// TwinCAT 3 PLC project Example
// ProgramVersion: 3.1.4026.16
// libraries:
//   Tc2_Standard, * (Beckhoff Automation GmbH)
//   Tc2_System, * (Beckhoff Automation GmbH)
//   Tc2_Utilities, * (Beckhoff Automation GmbH)
//   VisuDialogs, * (System)
//   StageCore, * (_)
//   StageUtils, * (_)
// project tree:
//   / GlobalTextList.TcGTLO, PlcTask.TcTTO (not stored), Visualization Manager.TcVMO (not stored), VISU_TASK.TcTTO (not stored)
//   Heating/Ctx/ Heating_Ctx_Hmi.TcPOU, Heating_Ctx_Io.TcDUT (not stored), Heating_Ctx_Priv.TcPOU, Heating_Ctx_States.TcPOU
//   Heating/Ctx/Io/ Heating_Ctx_Io_In.TcDUT, Heating_Ctx_Io_Out.TcDUT (not stored)
//   Heating/ Heating.TcPOU, Heating_Ctx.TcPOU (not stored)
//   Heating/Receivers/ Heating_OnRequest.TcPOU
//   Heating/State/ Heating_State.TcPOU, Heating_State_Enabled.TcPOU, Heating_State_Disabled.TcPOU, Heating_State_Heatup.TcPOU, Heating_State_HeatingRoom.TcPOU, Heating_State_Safety.TcPOU, Heating_State_Fault.TcPOU
//   MAIN/ CST.TcGVL, COL.TcGVL, MAIN.TcPOU, MAIN.TcVIS, SIM.TcGVL
//   MAIN/SIM/ SimulationGlobalParameters.TcDUT, Tick.TcPOU, ValveSim.TcPOU
//   Room/Rooms/ ReceptionRoom.TcPOU, BaseRoom.TcPOU, StandardRoom.TcPOU
//   Room/ IArgToIRoom.TcPOU (not stored), I_Room.TcIO (not stored), Room_Ctx.TcPOU
//   Room/Ctx/ Room_Ctx_Hmi.TcPOU, Room_Ctx_Io.TcDUT, Room_Ctx_Priv.TcPOU (not stored), Room_Ctx_States.TcPOU
//   Room/Receivers/ Room_OnSystemEvent.TcPOU
//   Room/State/DemandHeating/ Room_State_DemandHeating.TcPOU, Room_State_DemandHeating_Hmi.TcPOU (not stored)
//   Room/State/LowTemperature/ Room_State_LowTemperature_Hmi.TcPOU (not stored), Room_State_LowTemperature.TcPOU
//   Room/State/ _Room_State.TcPOU, Room_State_Idle.TcPOU, Room_State_Fault.TcPOU, Room_State_Disabled.TcPOU
//   Room/UI/ Room_UiLogic.TcPOU
//   Safety/ Safety.TcPOU, Safety_Hmi.TcPOU
//   _UI/ UI_Heating.TcVIS, UI_Safety.TcVIS, UI_Room.TcVIS, UI_Sim.TcVIS, UI_Temp.TcVIS, UI_Demand.TcVIS (not stored)
// (motion and I/O tree: see PLC project stageutils)
// real-time tasks:
//   TASK Example: cycle T#10ms, priority 20, ADS port 350
//   TASK Test: cycle T#10ms, priority 21, ADS port 351
//   TASK VISU_TASK: cycle T#200000us, priority 30, ADS port 352

// ---- Heating/Ctx/Io/Heating_Ctx_Io_In.TcDUT
TYPE Heating_Ctx_Io_In :
STRUCT
	bPumpOverload	: BOOL;
	bBurnerOverload	: BOOL;
	
	rBoilerTemp		: REAL;
	rBoilerPressure	: REAL;
END_STRUCT
END_TYPE

// ---- MAIN/SIM/SimulationGlobalParameters.TcDUT
TYPE SimulationGlobalParameters :
STRUCT
	// Simulation parameter
	nTick							: UDINT := 1000; // ms
	bToggleSim						: BOOL;	

	// Heating system parameters
	rSystemTemperatureRisePerBurner	: REAL := 2.00;   // degC/tick
	rSystemTemperatureDropPassive	: LREAL := -0.01;  // degC/tick
	rSystemTemperatureDropPerHeater	: LREAL := -0.01;  // degC/tick per heater
	
	bToggleSystemTemperatureRise	: BOOL := FALSE;
	rSystemTemperatureRise			: LREAL := 0.2;
	
	bToggleSystemTemperatureFall	: BOOL := FALSE;
	rSystemTemperatureFall			: LREAL := 0.2;
	
	bToggleSystemPressureRise		: BOOL := FALSE;
	rSystemPressureRise				: LREAL := 0.10;   // bar/tick
	
	bToggleSystemPressureFall		: BOOL := FALSE;
	rSystemPressureFall				: LREAL := -0.10;   // bar/tick
	
	// Room parameters
	rRoomTemperaturePassiveDrop		: LREAL := -0.05;  // degC/tick
	rRoomTemperatureRisePerHeater	: LREAL := 0.50;   // degC/tick
	
	// Valve fault
	bToggleValveFault				: BOOL;
	
END_STRUCT
END_TYPE

// ---- Room/Ctx/Room_Ctx_Io.TcDUT
TYPE Room_Ctx_Io :
STRUCT
	bOpenValves			: BOOL;
END_STRUCT
END_TYPE

// ---- MAIN/CST.TcGVL
{attribute 'qualified_only'}
VAR_GLOBAL CONSTANT
	MAX_ROOM		: UDINT := 15;
	MAX_ESTOP		: UDINT := 2;
END_VAR

// ---- MAIN/COL.TcGVL
{attribute 'qualified_only'}
VAR_GLOBAL CONSTANT
{warning disable C0228}	// Disable warning: No initial value for variable ...
	RED			: Color(255, 0, 0, 255);
	BLACK		: Color(0, 0, 0, 255);
	ORANGE		: Color(255, 160, 0, 255);
	WHITE		: Color(255, 255, 255, 255);
	INVISIBLE	: Color(0, 0, 0, 0);
{warning restore C0228}
END_VAR

// ---- MAIN/SIM.TcGVL
{attribute 'qualified_only'}
VAR_GLOBAL PERSISTENT
	param			: SimulationGlobalParameters;
END_VAR

VAR_GLOBAL
	bTick				: BOOL;	

	rSystemTemperature	: REAL := 60;
	rSystemPressure		: REAL := 1;
	bFlow				: BOOL;
END_VAR

// ---- Heating/Ctx/Heating_Ctx_Hmi.TcPOU
FUNCTION_BLOCK Heating_Ctx_Hmi
VAR_INPUT
	sStatusText				: Str;
	sErrorText				: Str;
	nStatusColor			: Color;
	
	bButton					: BOOL;
	sButtonText				: Str;
	nButtonColor			: Color;	
END_VAR
VAR_OUTPUT PERSISTENT
	rMaxPressure			: REAL := 2.0; // bar
	rMinPressure			: REAL := 0.2; // bar
	
	rMaxTemperature			: REAL := 65.0; // °C
	rStdTemperature			: REAL := 60.0; // °C
	rMinTemperature			: REAL := 55.0; // °C
END_VAR

END_FUNCTION_BLOCK

// ---- Heating/Ctx/Heating_Ctx_Priv.TcPOU
FUNCTION_BLOCK Heating_Ctx_Priv
VAR_INPUT
	iActiveRoom		: I_Room;
END_VAR
VAR_OUTPUT
	iOnEnable		: I_SignalEmit;
	
	iQueue			: I_MutArgQueue;
END_VAR

END_FUNCTION_BLOCK

// ---- Heating/Ctx/Heating_Ctx_States.TcPOU
FUNCTION_BLOCK Heating_Ctx_States
VAR_OUTPUT
	iMgr			: I_StateManager;
	
	iSafety			: I_State;
	iFault			: I_State;
	iDisable		: I_State;
	iEnable			: I_State;
	iPump			: I_State;
	iHeatup			: I_State;
	
END_VAR

END_FUNCTION_BLOCK

// ---- Heating/Heating.TcPOU
FUNCTION_BLOCK Heating 
VAR_GENERIC CONSTANT
	ROOM_CAP		: UDINT := 20;
END_VAR

IMPLEMENTS I_Execute, I_Init
VAR_INPUT
	bPumpOverload	: BOOL;
	bBurnerOverload	: BOOL;

	rBoilerTemp		: LREAL := 60;
	rBoilerPressure	: LREAL := 1;
END_VAR
VAR_OUTPUT
	bPump			: BOOL;
	bBurner			: BOOL;
END_VAR
VAR
	_init			: Init(THIS^);
	_exe			: Execute(THIS^);
	_ctx			: Heating_Ctx;
	_tonPump		: TON;
	_tonBurner		: TON;	

	_entityStart	: EntityStart;
	_tag			: Tag := (Option := 'Heating');

	_smgr			: StateManager := (Proxy := _ctx.state.iMgr);
	
	_disabled		: Heating_State_Disabled(_ctx) := (Proxy := _ctx.state.iDisable);
	_safety         : Heating_State_Safety(_ctx) := (Proxy := _ctx.state.iSafety);
	_fault          : Heating_State_Fault(_ctx) := (Proxy := _ctx.state.iFault);
	_enabled        : Heating_State_Enabled(_ctx) := (Proxy := _ctx.state.iEnable);
	_pumping        : Heating_State_HeatingRoom(_ctx) := (Proxy := _ctx.state.iHeating);
	_heatup         : Heating_State_Heatup(_ctx) := (Proxy := _ctx.state.iHeatup);

	_enableEvent	: Signal := (Proxy := _ctx.priv.iOnEnable);
	_onRequestCall	: Heating_OnRequest(_ctx);
	_onRequest		: Receiver(_onRequestCall);
	
	_queue			: ArgQueue<ROOM_CAP> := (MutProxy := _ctx.priv.iQueue);
	
	_entityEnd		: EntityEnd;
END_VAR

METHOD Execute
VAR_INPUT
	nPhase: INT := 0;
END_VAR
// Inputs
_ctx.io.in.bBurnerOverload := bBurnerOverload;
_ctx.io.in.bPumpOverload := bPumpOverload;
_ctx.io.in.rBoilerPressure := rBoilerPressure;
_ctx.io.in.rBoilerTemp := rBoilerTemp;

// Outputs
_tonPump(IN := _ctx.io.out.bPump, PT := T#2S, Q => bPump);
_tonBurner(IN := _ctx.io.out.bBurner, PT := T#2S, Q => bBurner);

// SIMULATION

IF NOT sim.bTick THEN
	RETURN;
END_IF

// System temperature
IF bBurner THEN
	sim.rSystemTemperature := sim.rSystemTemperature + Sim.param.rSystemTemperatureRisePerBurner * Math.Random();
END_IF
sim.rSystemTemperature := sim.rSystemTemperature + Sim.param.rSystemTemperatureDropPassive * Math.Random();

IF sim.param.bToggleSystemTemperatureRise THEN
	sim.rSystemTemperature := sim.rSystemTemperature + Sim.param.rSystemTemperatureRise;
END_IF
IF sim.param.bToggleSystemTemperatureFall THEN
	sim.rSystemTemperature := sim.rSystemTemperature + Sim.param.rSystemTemperatureFall;
END_IF

IF sim.rSystemTemperature < 0 THEN
	sim.rSystemTemperature := 0;
ELSIF sim.rSystemTemperature > 100 THEN
	sim.rSystemTemperature := 100;
END_IF

sim.bFlow := bPump;

// System Pressure
IF sim.param.bToggleSystemPressureRise THEN
	sim.rSystemPressure := sim.rSystemPressure + Sim.param.rSystemPressureRise;
END_IF
IF sim.param.bToggleSystemPressureFall THEN
	sim.rSystemPressure := sim.rSystemPressure + Sim.param.rSystemPressureFall;
END_IF

IF sim.rSystemPressure < 0 THEN
	sim.rSystemPressure := 0;
ELSIF sim.rSystemPressure > 10 THEN
	sim.rSystemPressure := 10;
END_IF

// Write IO

rBoilerTemp := sim.rSystemTemperature;
rBoilerPressure := sim.rSystemPressure;
END_METHOD

METHOD Init
VAR_INPUT
	nPhase: INT;
END_VAR
_smgr.Request(_disabled);
END_METHOD

END_FUNCTION_BLOCK

// ---- Heating/State/Heating_State_Disabled.TcPOU
FUNCTION_BLOCK Heating_State_Disabled EXTENDS Heating_State
VAR_INPUT
END_VAR
VAR_OUTPUT
END_VAR
VAR
END_VAR

METHOD PROTECTED OnEntry
_ctx.hmi.sStatusText := 'Heating disabled!';
_ctx.hmi.nStatusColor := COL.BLACK.Raw;

_ctx.hmi.sButtonText := 'Press to ENABLE!';
_ctx.hmi.nButtonColor := COL.BLACK.Raw;

_ctx.io.out.bBurner := FALSE;
_ctx.io.out.bPump := FALSE;

_ctx.priv.iQueue.Clear();
END_METHOD

METHOD PROTECTED OnExecute
IF _ctx.hmi.bButton THEN
	_ctx.hmi.bButton := FALSE;
	_ctx.state.iMgr.Request(_ctx.state.iEnable);
END_IF
END_METHOD

END_FUNCTION_BLOCK

// ---- Heating/State/Heating_State.TcPOU
FUNCTION_BLOCK ABSTRACT Heating_State EXTENDS State
VAR
	_ctx			: REFERENCE TO Heating_Ctx;
END_VAR

(*FB_Init is always available implicitly and it is used primarily for initialization.
The return value is not evaluated. For a specific influence, you can also declare the
methods explicitly and provide additional code there with the standard initialization
code. You can evaluate the return value.*)
METHOD FB_Init : BOOL
VAR_INPUT
	(* TRUE: the retain variables are initialized (reset warm / reset cold)*)
	bInitRetains	: BOOL;
	(* TRUE: the instance will be copied to the copy code afterward (online change)*)
	bInCopyCode	: BOOL;
	iEntity	: Core.I_Entity;
	ctx		: REFERENCE TO Heating_Ctx;
END_VAR
_ctx REF= ctx;
END_METHOD

END_FUNCTION_BLOCK

// ---- Heating/State/Heating_State_Safety.TcPOU
FUNCTION_BLOCK Heating_State_Safety EXTENDS Heating_State IMPLEMENTS I_Callable, I_Init
VAR
	_init					: Init(THIS^);
	_safetyRec				: Receiver(THIS^);
	_bSafetyStopActive			: BOOL;
END_VAR

METHOD Call
VAR_INPUT
	iArg		: StageCore.I_Arg;
END_VAR
VAR
	_iSafeModeOn: I_BoolArg;
END_VAR
IF IsOk(IArgToIBoolArg(iArg, _iSafeModeOn)) THEN
	IF _iSafeModeOn.Get THEN
		_bSafetyStopActive := TRUE;
		_ctx.state.iMgr.Request(_ctx.state.iSafety);
	ELSE
		_bSafetyStopActive := FALSE;
		_ctx.state.iMgr.Request(_ctx.state.iDisable);
	END_IF
END_IF
END_METHOD

METHOD PROTECTED CanDeactivate : BOOL
CanDeactivate := NOT _bSafetyStopActive;
END_METHOD

METHOD Init
VAR_INPUT
	nPhase: INT;
END_VAR
VAR
	i			: Iter(1);
	_r			: Result;
	
	_iEntity	: I_Entity;
	_iSignal	: I_Signal;
	
	
END_VAR
WHILE IsOk(GetEntity(i.Next(), _iEntity)) DO
	IF IsOk(GetSignal(_iEntity, '*._safetyEvent', _iSignal)) THEN
		IF IsFail(_iSignal.Pair(_safetyRec), nOut => _r) THEN
			DebugMsg(_iSignal, CONCAT('Could not be paired! Error code: ', TO_STRING(_r)));
		END_IF
		
		RETURN;
	END_IF
END_WHILE

DebugMsg(THIS^, CONCAT('_safetyRec not paired! Error code: ', TO_STRING(_r)));
END_METHOD

METHOD PROTECTED OnEntry
_ctx.hmi.sStatusText := 'Safety engaged! Check safety system...';
_ctx.hmi.nStatusColor := COL.RED.Raw;

_ctx.hmi.sButtonText := '';
_ctx.hmi.nButtonColor := COL.INVISIBLE.Raw;

_ctx.io.out.bBurner := FALSE;
_ctx.io.out.bPump := FALSE;

_ctx.priv.iQueue.Clear();
END_METHOD

END_FUNCTION_BLOCK

// ---- Safety/Safety.TcPOU
FUNCTION_BLOCK Safety 
VAR_GENERIC CONSTANT
	ESTOP_CAP		: UDINT := 2;
END_VAR
IMPLEMENTS I_Execute
VAR_INPUT
	bSafetyOk		: BOOL;
	bEStopActive	: ARRAY[1..ESTOP_CAP] OF BOOL;
END_VAR
VAR_OUTPUT
	bSafetyRun		: BOOL;
	bErrAck			: BOOL;
END_VAR
VAR
	_exe			: Execute(THIS^);
	_hmi			: Safety_Hmi<ESTOP_CAP>;
	_nStep			: USINT;
	_tonTimeout		: TON;	

	_entityStart		: EntityStart;
	_tag				: Tag := (Option := 'Safety');

	_safetyEvent		: Signal;
	_bSafetyStopActive	: BoolArg(FALSE);
	
	_entityEnd			: EntityEnd;
END_VAR

METHOD Execute
VAR_INPUT
	nPhase: INT;
END_VAR
VAR
	i			: UDINT;
END_VAR
FOR i := 1 TO ESTOP_CAP DO
	_hmi.bEStopActive[i] := bESTopActive[i];
END_FOR


CASE _nStep OF
	0: // Fault Init
		_bSafetyStopActive.OpSet(TRUE);
		_safetyEvent.Emit(_bSafetyStopActive);
		bSafetyRun	:= FALSE;
		
		_nStep := 1;
		
		_hmi.bHideReset := TRUE;
		_hmi.nStatusColor := COL.RED.Raw;
		_hmi.sStatusText := 'Safety Stop Activated!';

	1: // Fault
		_hmi.bHideReset := NOT bSafetyOk;
		IF bSafetyOk AND _hmi.bReset THEN
			_hmi.bReset := FALSE;
			
			_nStep := 2;
		END_IF

	2: // Reset init
		bSafetyRun	:= TRUE;
		
		_nStep		:= 3;
		
		_hmi.bHideReset := TRUE;
		_hmi.nStatusColor := COL.RED.Raw;
		_hmi.sStatusText := 'Reset in progress...';
		
	3: // Reset
	
		bErrAck		:= TRUE;
		
		_tonTimeout(IN := TRUE, PT := T#5S);
		
		IF bSafetyOk THEN
			_tonTimeout(IN := FALSE);
			_nStep := 4;
		ELSIF _tonTimeout.Q THEN
			_tonTimeout(IN := FALSE);
			_nStep := 0;
		END_IF	

	4:	// Op Init
		bErrAck		:= FALSE;
	
		_bSafetyStopActive.OpSet(FALSE);
		_safetyEvent.Emit(_bSafetyStopActive);
		_nStep := 5;
		
		_hmi.bHideReset := TRUE;
		_hmi.nStatusColor := COL.BLACK.Raw;
		_hmi.sStatusText := 'Safety OK!';

	5:	// Op
		IF NOT bSafetyOk THEN
			_nStep := 0;
		END_IF
END_CASE
END_METHOD

END_FUNCTION_BLOCK

// ---- Safety/Safety_Hmi.TcPOU
FUNCTION_BLOCK Safety_Hmi
VAR_GENERIC CONSTANT
	ESTOP_CAP		: UDINT := 4;
END_VAR

VAR_INPUT
	bEStopActive	: ARRAY[1..ESTOP_CAP] OF BOOL;
	
	sStatusText		: Str;
	nStatusColor	: Color;
	
	bReset			: BOOL;
	bHideReset		: BOOL;
END_VAR

END_FUNCTION_BLOCK

// ---- Heating/State/Heating_State_Fault.TcPOU
FUNCTION_BLOCK Heating_State_Fault EXTENDS Heating_State IMPLEMENTS I_Execute
VAR
	_exe		: Execute(THIS^);
END_VAR

METHOD Execute
VAR_INPUT
	nPhase: INT;
END_VAR
VAR
	cmp			: TagCmp;
	bFault		: BOOL;
END_VAR
IF _ctx.io.in.bBurnerOverload THEN
	bFault := TRUE;
END_IF

IF _ctx.io.in.bPumpOverload THEN
	bFault := TRUE;
END_IF

IF _ctx.io.in.rBoilerPressure > _ctx.hmi.rMaxPressure THEN
	bFault := TRUE;
END_IF

IF _ctx.io.in.rBoilerPressure < _ctx.hmi.rMinPressure THEN
	bFault := TRUE;
END_IF

IF _ctx.io.in.rBoilerTemp > _ctx.hmi.rMaxTemperature THEN
	bFault := TRUE;
END_IF

IF cmp.Set(_ctx.state.iMgr.Current.Tag).Match(_ctx.state.iFault.Tag).Match(_ctx.state.iSafety.Tag).IsTrue() THEN
	bFault := FALSE;
END_IF

IF NOT bFault THEN
	RETURN;
END_IF

_ctx.state.iMgr.Request(_ctx.state.iFault);
END_METHOD

METHOD PROTECTED OnEntry
IF _ctx.io.in.bBurnerOverload THEN
	_ctx.hmi.sErrorText := 'Caused by burner overload!';
ELSIF _ctx.io.in.bPumpOverload THEN
	_ctx.hmi.sErrorText := 'Caused by pump overload!';
ELSIF _ctx.io.in.rBoilerPressure > _ctx.hmi.rMaxPressure THEN
	_ctx.hmi.sErrorText := 'Caused by boiler overpressure!';
ELSIF _ctx.io.in.rBoilerPressure < _ctx.hmi.rMinPressure THEN
	_ctx.hmi.sErrorText := 'Caused by boiler underpressure!';
ELSIF _ctx.io.in.rBoilerTemp > _ctx.hmi.rMaxTemperature THEN
	_ctx.hmi.sErrorText := 'Caused by boiler overheat!';
END_IF

_ctx.hmi.sStatusText := CONCAT('Fault: ', _ctx.hmi.sErrorText);

_ctx.hmi.nStatusColor := COL.RED.Raw;

_ctx.hmi.sButtonText := 'Press to RESET';
_ctx.hmi.nButtonColor := COL.INVISIBLE.Raw;

_ctx.io.out.bBurner := FALSE;
_ctx.io.out.bPump := FALSE;

_ctx.priv.iQueue.Clear();
END_METHOD

METHOD PROTECTED OnExecute
VAR
	bFault : BOOL;
END_VAR
IF _ctx.io.in.bBurnerOverload THEN
	bFault := TRUE;
END_IF

IF _ctx.io.in.bPumpOverload THEN
	bFault := TRUE;;
END_IF

IF _ctx.io.in.rBoilerPressure > _ctx.hmi.rMaxPressure THEN
	bFault := TRUE;;
END_IF

IF _ctx.io.in.rBoilerPressure < _ctx.hmi.rMinPressure THEN
	bFault := TRUE;;
END_IF

IF _ctx.io.in.rBoilerTemp > _ctx.hmi.rMaxTemperature THEN
	bFault := TRUE;;
END_IF

IF _ctx.hmi.bButton AND NOT bFault THEN
	_ctx.hmi.bButton := FALSE;
	_ctx.state.iMgr.Request(_ctx.state.iDisable);
ELSIF NOT bFault THEN
	_ctx.hmi.nButtonColor := COL.BLACK.Raw;	
ELSE
	_ctx.hmi.nButtonColor := COL.INVISIBLE.Raw;	
	_ctx.hmi.bButton := FALSE;
END_IF
END_METHOD

END_FUNCTION_BLOCK

// ---- Heating/State/Heating_State_Enabled.TcPOU
FUNCTION_BLOCK Heating_State_Enabled EXTENDS Heating_State
VAR_INPUT
END_VAR
VAR_OUTPUT
END_VAR
VAR
END_VAR

METHOD PROTECTED OnEntry
_ctx.hmi.sStatusText := 'Heating enabled: Waiting for requests...';
_ctx.hmi.nStatusColor := COL.BLACK.Raw;

_ctx.hmi.sButtonText := 'Press to DISABLE!';
_ctx.hmi.nButtonColor := COL.BLACK.Raw;

_ctx.io.out.bBurner := FALSE;
_ctx.io.out.bPump := FALSE;

IF _ctx.state.iMgr.Current = _ctx.state.iDisable THEN
	_ctx.priv.iOnEnable.Emit();
END_IF
END_METHOD

METHOD PROTECTED OnExecute
VAR
	_iRoomArg		: I_Arg;
END_VAR
IF _ctx.hmi.bButton THEN
	_ctx.hmi.bButton := FALSE;
	_ctx.state.iMgr.Request(_ctx.state.iDisable);
	
ELSIF _ctx.io.in.rBoilerTemp < _ctx.hmi.rMinTemperature THEN
	_ctx.state.iMgr.Request(_ctx.state.iHeatup);
	
ELSIF IsOk(_ctx.priv.iQueue.Pop(iArg => _iRoomArg)) THEN
	IF IsOk(IArgToIRoom(_iRoomArg, iDest => _ctx.priv.iActiveRoom)) THEN
		IF _ctx.priv.iActiveRoom.IsActive THEN
			_ctx.state.iMgr.Request(_ctx.state.iHeating);
		END_IF
	ELSE
		_ctx.hmi.sErrorText := 'Room Queue - Incorrect iRoomArg!';
	END_IF
END_IF
END_METHOD

END_FUNCTION_BLOCK

// ---- Heating/State/Heating_State_HeatingRoom.TcPOU
FUNCTION_BLOCK Heating_State_HeatingRoom EXTENDS Heating_State
VAR CONSTANT
	EXIT_STEP		: USINT := 7;
	READY_STEP		: USINT := 8;
END_VAR
VAR
	_nStep		: USINT;
	_tonTimeout	: TON;
	_sErrMsg	: Str;
	_iNextState : I_State;
END_VAR

METHOD PROTECTED CanActivate : BOOL
CanActivate :=  _ctx.state.iMgr.Current = _ctx.state.iEnable;
END_METHOD

METHOD PROTECTED OnEntry
VAR
	strb			: Strb;
END_VAR
_ctx.hmi.sStatusText := strb.Append('Heating enabled: Pumping to room ')
							.Append(UDINT_TO_STRING(_ctx.priv.iActiveRoom.Id))
							.Append('...')
							.Read();
							
_ctx.hmi.nStatusColor := COL.BLACK.Raw;

_ctx.hmi.sButtonText := 'Press to DISABLE!';
_ctx.hmi.nButtonColor := COL.BLACK.Raw;

_ctx.io.out.bBurner := FALSE;
_ctx.io.out.bPump := FALSE;

_nStep := 0;
_tonTimeout(IN := FALSE);

_iNextState := _ctx.state.iEnable;
END_METHOD

METHOD PROTECTED OnExecute
VAR
	strb		: Strb;
END_VAR
IF _ctx.priv.iActiveRoom = 0 THEN
	_iNextState := _ctx.state.iFault;	

	_nStep := EXIT_STEP;
	_ctx.hmi.sErrorText := 'HeatingRoom - Incorrect iActiveRoom value!';
ELSIF _ctx.hmi.bButton THEN
	_ctx.hmi.bButton := FALSE;
	_iNextState := _ctx.state.iDisable;
	
	_nStep := 4;
ELSIF _tonTimeout.Q THEN
	_ctx.priv.iActiveRoom.GoFault(strb.Set('Timeout on: ').Append(_sErrMsg).Read());
	
	_nStep := EXIT_STEP;
ELSIF _nStep < 4 AND_THEN NOT _ctx.priv.iActiveRoom.IsActive THEN
	_iNextState := _ctx.state.iEnable;	

	_nStep := 4;
END_IF

IF _ctx.priv.iActiveRoom <> 0 THEN
	_tonTimeout(IN := TRUE, PT := _ctx.priv.iActiveRoom.Timeout);
END_IF

CASE _nStep OF
	0:
		_sErrMsg := 'Valve opening!';
		_ctx.priv.iActiveRoom.GoHeat();
		_nStep := 1;
		
	1:
		IF _ctx.priv.iActiveRoom.IsOpen THEN
			_nStep := 2;
		END_IF
	2:	
		
		_ctx.io.out.bPump := TRUE;
		_nStep := 3;
	3:
		_sErrMsg := 'Heating!';
		IF _ctx.priv.iActiveRoom.IsReady THEN
			_nStep := 4;
		END_IF
	4:	
		_ctx.io.out.bPump := FALSE;
		_nStep := 5;
	5:
		_sErrMsg := 'Valve closing!';
		_ctx.priv.iActiveRoom.GoIdle();
		_nStep := 6;
	6:
		IF _ctx.priv.iActiveRoom.IsClosed THEN
			_nStep := EXIT_STEP;
		END_IF
	7:
		IF _iNextState <> 0 THEN
			_ctx.state.iMgr.Request(_iNextState);
		ELSE
			_ctx.hmi.sErrorText := 'HeatingRoom - Incorrect _iNextState value!';
			_ctx.state.iMgr.Request(_ctx.state.iFault);
		END_IF
		
		_nStep := READY_STEP;
END_CASE
END_METHOD

(*
Executed when the state transitions to another state.  
Provides a hook for defining cleanup or transition-specific behavior.
*)
METHOD PROTECTED OnExit
IF _ctx.priv.iActiveRoom <> 0 THEN
	_ctx.priv.iActiveRoom.GoIdle();
END_IF
END_METHOD

END_FUNCTION_BLOCK

// ---- Heating/State/Heating_State_Heatup.TcPOU
FUNCTION_BLOCK Heating_State_Heatup EXTENDS Heating_State
VAR_INPUT
END_VAR
VAR_OUTPUT
END_VAR
VAR
END_VAR

METHOD CanActivate : BOOL
CanActivate :=  _ctx.state.iMgr.Current = _ctx.state.iEnable;
END_METHOD

METHOD OnEntry
_ctx.hmi.sStatusText := 'Heating enabled: Heating up...';
_ctx.hmi.nStatusColor := COL.BLACK.Raw;

_ctx.hmi.sButtonText := 'Press to DISABLE!';
_ctx.hmi.nButtonColor := COL.BLACK.Raw;

_ctx.io.out.bBurner := TRUE;
_ctx.io.out.bPump := TRUE;
END_METHOD

METHOD OnExecute
IF _ctx.hmi.bButton THEN
	_ctx.hmi.bButton := FALSE;
	_ctx.state.iMgr.Request(_ctx.state.iDisable);
	
ELSIF _ctx.io.in.rBoilerTemp >= _ctx.hmi.rStdTemperature THEN
	_ctx.state.iMgr.Request(_ctx.state.iEnable);
END_IF
END_METHOD

END_FUNCTION_BLOCK

// ---- Heating/Receivers/Heating_OnRequest.TcPOU
FUNCTION_BLOCK Heating_OnRequest IMPLEMENTS I_Callable
VAR
	_ctx			: REFERENCE TO Heating_Ctx;
END_VAR

METHOD Call
VAR_INPUT
	iArg				: Core.I_Arg;
END_VAR
VAR
	_iRoom				: I_Room;
END_VAR
IF IsOk(IArgToIRoom(iArg, iDest => _iRoom)) THEN
	_ctx.priv.iQueue.Push(_iRoom);
END_IF
END_METHOD

//FB_Init is always available implicitly and it is used primarily for initialization.
//The return value is not evaluated. For a specific influence, you can also declare the
//methods explicitly and provide additional code there with the standard initialization
//code. You can evaluate the return value.
METHOD FB_Init: BOOL
VAR_INPUT
    bInitRetains: BOOL; // TRUE: the retain variables are initialized (reset warm / reset cold)
    bInCopyCode: BOOL;  // TRUE: the instance will be copied to the copy code afterward (online change)

	ctx			: REFERENCE TO Heating_Ctx;   
END_VAR
_ctx REF= ctx;
END_METHOD

END_FUNCTION_BLOCK

// ---- MAIN/MAIN.TcPOU
PROGRAM MAIN
VAR
	safety				: Safety<CST.MAX_ESTOP>;
	heating				: Heating<CST.MAX_ROOM>;
	
	stdRoom				: ARRAY[1..3] OF StandardRoom;
	reception			: ReceptionRoom;

	dbgInfo				: DebugInfo;
	rtTick				: R_TRIG;
END_VAR

rtTick(CLK :=  Tick(sim.param.nTick), Q => sim.bTick);
sim.bTick := sim.bTick AND sim.param.bToggleSim;

Runtime();

END_PROGRAM

// ---- Room/Rooms/StandardRoom.TcPOU
FUNCTION_BLOCK StandardRoom EXTENDS BaseRoom
VAR_INPUT
	rTemperature	: LREAL := 20.0 + Math.Random();
END_VAR
VAR    	
    // Entity
    _entityExtend	: EntityExtend(_entityStart);
	
    _lowTemperature : Room_State_LowTemperature(_ctx, rTemperature);
    _demand         : Room_State_DemandHeating(_ctx);
   
    _entityEnd2		: EntityEnd;
END_VAR

METHOD Execute
SUPER^.Execute();

// Simulation
IF NOT sim.bTick THEN
	RETURN;
END_IF

IF bInletValve AND bOutletValve THEN
	rTemperature := rTemperature + sim.param.rRoomTemperatureRisePerHeater * Math.Random();
END_IF

rTemperature := rTemperature + sim.param.rRoomTemperaturePassiveDrop * Math.Random();

IF rTemperature < 0 THEN
	rTemperature := 0;
ELSIF rTemperature > 100 THEN
	rTemperature := 100;
END_IF
END_METHOD

END_FUNCTION_BLOCK

// ---- Room/Rooms/BaseRoom.TcPOU
FUNCTION_BLOCK BaseRoom IMPLEMENTS I_Execute, I_Init
VAR_INPUT	
	bInletValveIsClosed	: BOOL;
	bInletValveIsOpen	: BOOL;
	
	bOutletValveIsClosed: BOOL;
	bOutletValveIsOpen	: BOOL;
END_VAR
VAR_OUTPUT
	bInletValve		: BOOL;
	bOutletValve	: BOOL;
END_VAR
VAR    
    // Initialization and execution logic
    _init           : Init(THIS^);
    _exe            : Execute(THIS^);
    _ctx            : Room_Ctx;
	
	// UI Logic
    _uiLogic        : Room_UiLogic(_ctx);
	
    // Simulation
    _inletSim       : ValveSim(bInletValve, bInletValveIsOpen, bInletValveIsClosed);
    _outletSim      : ValveSim(bOutletValve, bOutletValveIsOpen, bOutletValveIsClosed);	
	
	
    // Entity
    _entityStart    : EntityStart;
	
    _tag            : Tag := (Option := CONCAT('Room_', UDINT_TO_STRING(_ctx.Id)));
    
    // State Manager
    _smgr           : StateManager := (Proxy := _ctx.state.iMgr);
    
    // States
    _disabled       : Room_State_Disabled(_ctx) := (Proxy := _ctx.state.iDisable);
    _fault          : Room_State_Fault(_ctx) := (Proxy := _ctx.state.iFault);
    _idle           : Room_State_Idle(_ctx) := (Proxy := _ctx.state.iIdle);
	
	// Receiver
    _onSystemEvent  : Room_OnSystemEvent(_ctx);
    
    // Signal
    _requestEvent   : Signal := (Proxy := _ctx.priv.iRequestEvent);
   
    _entityEnd      : EntityEnd;
END_VAR

METHOD Execute
VAR_INPUT
	nPhase: INT;
END_VAR
// HMI

_ctx.hmi.sData := '';

// Inputs
_ctx.io.bValvesOpen := bInletValveIsOpen AND bOutletValveIsOpen;
_ctx.io.bValvesClosed := bInletValveIsClosed AND bOutletValveIsClosed;

// Outputs
bInletValve := _ctx.io.bOpenValves;
bOutletValve := _ctx.io.bOpenValves;

// Simulation
IF NOT sim.bTick THEN
	RETURN;
END_IF

IF bInletValve AND bOutletValve THEN
	sim.rSystemTemperature := sim.rSystemTemperature + sim.param.rSystemTemperatureDropPerHeater * Math.Random();
END_IF
END_METHOD

METHOD Init
VAR_INPUT
	nPhase: INT;
END_VAR
_smgr.Request(_idle);
END_METHOD

END_FUNCTION_BLOCK

// ---- Room/Room_Ctx.TcPOU
FUNCTION_BLOCK Room_Ctx
VAR_INPUT
	io		: Room_Ctx_Io; // different
	hmi		: Room_Ctx_Hmi; // the same
	state	: Room_Ctx_States; // the same
	priv	: Room_Ctx_Priv; // the same but different logic
END_VAR

END_FUNCTION_BLOCK

// ---- Room/Ctx/Room_Ctx_Hmi.TcPOU
FUNCTION_BLOCK Room_Ctx_Hmi
VAR_INPUT
	nId						: UDINT;	

	sStatusText				: Str;
	sErrorText				: Str;
	nStatusColor			: Color;
	
	sData					: Str;
	
	bDisable				: BOOL;
	sDisableText			: Str;
	
	bReset					: BOOL;
	bHideReset				: BOOL;
END_VAR
VAR_OUTPUT PERSISTENT
	nTimeout				: UDINT := 1;
END_VAR

END_FUNCTION_BLOCK

// ---- Room/Ctx/Room_Ctx_States.TcPOU
FUNCTION_BLOCK Room_Ctx_States
VAR_OUTPUT
	iMgr			: I_StateManager;
	
	iSystemOff		: I_State;
	iFault			: I_State;
	iDisable		: I_State;
	iIdle			: I_State;
END_VAR

END_FUNCTION_BLOCK

// ---- Room/UI/Room_UiLogic.TcPOU
FUNCTION_BLOCK Room_UiLogic IMPLEMENTS I_Execute
VAR_INPUT
END_VAR
VAR_OUTPUT
END_VAR
VAR
	_exe			: Execute(THIS^);
	_ctx			: REFERENCE TO Room_Ctx;
	
	_bPrvDisable	: BOOL;
END_VAR

METHOD Execute
IF _bPrvDisable <> _ctx.hmi.bDisable THEN
	_bPrvDisable := _ctx.hmi.bDisable;
	
	IF _ctx.hmi.bDisable THEN
		_ctx.hmi.sDisableText := 'Press to ENABLE!';
	ELSE
		_ctx.hmi.sDisableText := 'Press to DISABLE!';
	END_IF	
END_IF
END_METHOD

//FB_Init is always available implicitly and it is used primarily for initialization.
//The return value is not evaluated. For a specific influence, you can also declare the
//methods explicitly and provide additional code there with the standard initialization
//code. You can evaluate the return value.
METHOD FB_Init: BOOL
VAR_INPUT
    bInitRetains: BOOL; // TRUE: the retain variables are initialized (reset warm / reset cold)
    bInCopyCode: BOOL;  // TRUE: the instance will be copied to the copy code afterward (online change)
	
	ctx			: REFERENCE TO Room_Ctx;
END_VAR
_ctx REF= ctx;

IF _ctx.hmi.bDisable THEN
	_ctx.hmi.sDisableText := 'Press to ENABLE!';
ELSE
	_ctx.hmi.sDisableText := 'Press to DISABLE!';
END_IF
END_METHOD

END_FUNCTION_BLOCK

// ---- MAIN/SIM/ValveSim.TcPOU
FUNCTION_BLOCK ValveSim IMPLEMENTS I_Execute
VAR
	_bInput		: REFERENCE TO BOOL;	
	_bIsOpen	: REFERENCE TO BOOL;
	_bIsClosed	: REFERENCE TO BOOL;	

	_exe		: Execute(THIS^);
	_ton		: TON := (PT := LREAL_TO_TIME(Math.Random() * 1000));
	_rt			: R_TRIG;
	_ft			: F_TRIG;
	_bInit		: BOOL := TRUE;
END_VAR

(*
If registered, this method will be executed cyclically.
*)
METHOD Execute
VAR_INPUT
	nPhase: INT;
END_VAR
_rt(CLK := _bInput);
_ft(CLK := _bInput);
IF _rt.Q OR _ft.Q OR _bInit THEN
	_ton.IN := TRUE;
	_bInit := FALSE;
END_IF

_ton();
IF _ton.Q AND SIM.param.bToggleValveFault THEN
	_ton(IN := FALSE);
	_bIsClosed := FALSE;
	_bIsOpen := FALSE;
	SIM.param.bToggleValveFault := FALSE;
ELSIF _ton.Q AND _bInput THEN
	_ton(IN := FALSE);
	_bIsOpen := TRUE;
	_bIsClosed := FALSE;
ELSIF _ton.Q AND NOT _bInput THEN
	_ton(IN := FALSE);
	_bIsOpen := FALSE;
	_bIsClosed := TRUE;	
END_IF
END_METHOD

//FB_Init is always available implicitly and it is used primarily for initialization.
//The return value is not evaluated. For a specific influence, you can also declare the
//methods explicitly and provide additional code there with the standard initialization
//code. You can evaluate the return value.
METHOD FB_Init: BOOL
VAR_INPUT
    bInitRetains: BOOL; // TRUE: the retain variables are initialized (reset warm / reset cold)
    bInCopyCode: BOOL;  // TRUE: the instance will be copied to the copy code afterward (online change) 

  	bInput		: REFERENCE TO BOOL;	
	bIsOpen		: REFERENCE TO BOOL;
	bIsClosed	: REFERENCE TO BOOL;	
END_VAR
_bInput REF= bInput;
_bIsOpen REF= bIsOpen;
_bIsClosed REF= bIsClosed;
END_METHOD

END_FUNCTION_BLOCK

// ---- Room/State/Room_State_Disabled.TcPOU
FUNCTION_BLOCK Room_State_Disabled EXTENDS _Room_State
VAR_INPUT
END_VAR
VAR_OUTPUT
END_VAR
VAR
END_VAR

METHOD OnEntry
_ctx.io.bOpenValves := FALSE;

_ctx.priv.bActive := FALSE;
_ctx.priv.bReady := FALSE;

_ctx.hmi.sStatusText := 'ROOM DISABLED!';
_ctx.hmi.nStatusColor := COL.RED.Raw;

_ctx.hmi.bHideReset := TRUE;
END_METHOD

METHOD OnExecute
IF NOT _ctx.hmi.bDisable THEN
	_ctx.state.iMgr.Request(_ctx.state.iIdle);
END_IF
END_METHOD

END_FUNCTION_BLOCK

// ---- Room/State/_Room_State.TcPOU
FUNCTION_BLOCK ABSTRACT _Room_State EXTENDS State
VAR
	_ctx	: REFERENCE TO Room_Ctx;
END_VAR

(*FB_Init is always available implicitly and it is used primarily for initialization.
The return value is not evaluated. For a specific influence, you can also declare the
methods explicitly and provide additional code there with the standard initialization
code. You can evaluate the return value.*)
METHOD FB_Init : BOOL
VAR_INPUT
	(* TRUE: the retain variables are initialized (reset warm / reset cold)*)
	bInitRetains	: BOOL;
	(* TRUE: the instance will be copied to the copy code afterward (online change)*)
	bInCopyCode	: BOOL;
	iEntity	: Core.I_Entity;
	ctx		: REFERENCE TO Room_Ctx;
END_VAR
_ctx REF= ctx;
END_METHOD

END_FUNCTION_BLOCK

// ---- Room/State/Room_State_Fault.TcPOU
FUNCTION_BLOCK Room_State_Fault EXTENDS _Room_State
VAR_INPUT
END_VAR
VAR_OUTPUT
END_VAR
VAR
END_VAR

METHOD PROTECTED OnEntry
_ctx.io.bOpenValves := FALSE;

_ctx.priv.bActive := FALSE;
_ctx.priv.bReady := FALSE;

_ctx.hmi.sStatusText := CONCAT('Fault: ', _ctx.hmi.sErrorText);
_ctx.hmi.nStatusColor := COL.RED.Raw;

_ctx.hmi.bHideReset := FALSE;
END_METHOD

METHOD PROTECTED OnExecute
IF _ctx.hmi.bReset THEN
	_ctx.hmi.bReset := FALSE;
	
	_ctx.state.iMgr.Request(_ctx.state.iIdle);
END_IF
END_METHOD

METHOD PROTECTED OnExit
_ctx.hmi.sErrorText := 'Undefined';
END_METHOD

END_FUNCTION_BLOCK

// ---- Room/State/Room_State_Idle.TcPOU
FUNCTION_BLOCK Room_State_Idle EXTENDS _Room_State
VAR_INPUT
END_VAR
VAR_OUTPUT
END_VAR
VAR
END_VAR

METHOD OnEntry
_ctx.io.bOpenValves := FALSE;

_ctx.priv.bActive := FALSE;
_ctx.priv.bReady := FALSE;

_ctx.hmi.sStatusText := 'Heating ON: Idle';
_ctx.hmi.nStatusColor := COL.BLACK.Raw;

_ctx.hmi.bHideReset := TRUE;
END_METHOD

METHOD OnExecute
IF _ctx.hmi.bDisable THEN
	_ctx.state.iMgr.Request(_ctx.state.iDisable);
END_IF
END_METHOD

END_FUNCTION_BLOCK

// ---- Room/Receivers/Room_OnSystemEvent.TcPOU
FUNCTION_BLOCK Room_OnSystemEvent IMPLEMENTS I_Init, I_Callable
VAR
	_init				: Init(THIS^);
	_onSystemEvent		: Receiver(THIS^);
	
	_bError				: BOOL;
	
	_iResumeEvent		: I_Signal;
	_iPauseEvent		: I_Signal;
	_iEnableEvent		: I_Signal;
	_iDisableEvent		: I_Signal;
	
	_ctx				: REFERENCE TO Room_Ctx;
END_VAR

METHOD PRIVATE _GetSignalAndPair
VAR_INPUT
	iEntity		: I_Entity;
	sToFind		: Str;
END_VAR
VAR_OUTPUT
	iSignal	: I_Signal;
END_VAR
VAR
	_r			: Result;
	strb		: Strb;
END_VAR
CASE GetSignal(iEntity, sToFind, iSignal) OF
	Ok:
		IF IsFail(iSignal.Pair(_onSystemEvent), nOut => _r) THEN
			_bError := TRUE;
			DebugMsg(iSignal, strb.Append('Cannot pair _systemRec with this signal! Error code: ').Append(INT_TO_STRING(_r)).Read());
		END_IF
	ELSE
		_bError := TRUE;
		DebugMsg(THIS^, strb.Append('Cannot pair _systemRec with a ').Append(sToFind).Append('!').Read());
		DebugMsg(iEntity, strb.Append(sToFind).Append(' not found!').Read());
END_CASE
END_METHOD

METHOD Call
VAR_INPUT
	iArg	: StageCore.I_Arg;
END_VAR
VAR
	cmp		: TagCmp;
	_iTag	: I_Tag;
END_VAR
IF _bError THEN
	_ctx.hmi.sErrorText := 'Incorrect receiver initialization!';
	_ctx.state.iMgr.Request(_ctx.state.iFault);
	RETURN;
END_IF

IF IsErr(IArgToITag(iArg, _iTag)) THEN
	_ctx.hmi.sErrorText := 'Incorrect call argument!';
	_ctx.state.iMgr.Request(_ctx.state.iFault);
	RETURN;
END_IF

cmp.Set(_iTag);
IF cmp.Match(_iEnableEvent.Tag).IsTrue() THEN
	IF _ctx.state.iMgr.Current = 0 THEN
		RETURN;
	END_IF

	cmp.Set(_ctx.state.iMgr.Current.Tag);
	IF cmp.Match(_ctx.state.iFault.Tag)
			.Match(_ctx.state.iDisable.Tag)
			.Match(_ctx.state.iIdle.Tag)
			.IsTrue() THEN
			
		RETURN;
	END_IF
	
	_ctx.priv.iRequestEvent.Emit(_ctx);
	
	RETURN;
END_IF
END_METHOD

//FB_Init is always available implicitly and it is used primarily for initialization.
//The return value is not evaluated. For a specific influence, you can also declare the
//methods explicitly and provide additional code there with the standard initialization
//code. You can evaluate the return value.
METHOD FB_Init: BOOL
VAR_INPUT
    bInitRetains: BOOL; // TRUE: the retain variables are initialized (reset warm / reset cold)
    bInCopyCode: BOOL;  // TRUE: the instance will be copied to the copy code afterward (online change)
	
	ctx			: REFERENCE TO Room_Ctx;
END_VAR
_ctx REF= ctx;
END_METHOD

METHOD Init
VAR_INPUT
	nPhase: INT;
END_VAR
VAR
	i			: Iter(1);
	_iEntity	: I_Entity;
END_VAR
WHILE IsOk(GetEntity(i.Next(), _iEntity)) DO
	IF IsFail(HasTagOption(_iEntity, 'Heating')) THEN
		CONTINUE;
	END_IF
	
	_GetSignalAndPair(_iEntity, '*._enableEvent', iSignal => _iEnableEvent);
	
	RETURN;
END_WHILE
END_METHOD

END_FUNCTION_BLOCK

// ---- Room/State/LowTemperature/Room_State_LowTemperature.TcPOU
FUNCTION_BLOCK Room_State_LowTemperature EXTENDS _Room_State IMPLEMENTS I_Execute, I_Init
VAR
	_init					: Init(THIS^);
	_exe					: Execute(THIS^);
	_hmi					: Room_State_LowTemperature_Hmi;
	_rTemperature			: REFERENCE TO LREAL;
END_VAR

METHOD PROTECTED CanActivate : BOOL
CanActivate := _ctx.state.iMgr.Current = _ctx.state.iIdle;
END_METHOD

METHOD Execute
VAR_INPUT
	nPhase: INT;
END_VAR
VAR
	_iSelf		: I_State := THIS^;
	_strb		: strb;
END_VAR
_strb.Set(_ctx.hmi.sData)
		.Append(' ')
		.Append(Strf.Fmt('%0.2f', F_LReal(_rTemperature)))
		.Append(' degC');

_ctx.hmi.sData := _strb.Read();

IF _ctx.state.iMgr.Current <> _ctx.state.iIdle THEN
	RETURN;
END_IF

IF _ctx.state.iMgr.Current = _iSelf THEN
	RETURN;
END_IF

IF _rTemperature < _hmi.rLowTemperature THEN
	_ctx.state.iMgr.Request(THIS^);
END_IF
END_METHOD

(*FB_Init is always available implicitly and it is used primarily for initialization.
The return value is not evaluated. For a specific influence, you can also declare the
methods explicitly and provide additional code there with the standard initialization
code. You can evaluate the return value.*)
METHOD FB_Init : BOOL
VAR_INPUT
	(* TRUE: the retain variables are initialized (reset warm / reset cold)*)
	bInitRetains	: BOOL;
	(* TRUE: the instance will be copied to the copy code afterward (online change)*)
	bInCopyCode	: BOOL;
	ctx				: REFERENCE TO Room_Ctx;
	rTemperature	: REFERENCE TO LREAL;
END_VAR
_rTemperature REF= rTemperature;
END_METHOD

METHOD Init
VAR_INPUT
	nPhase: INT;
END_VAR
VAR
	i			: Iter(1);
	_iEntity	: I_Entity;
	_iRec		: I_Receiver;
	_r			: Result;
	strb		: Strb;
END_VAR
WHILE IsOk(GetEntity(i.Next(), _iEntity)) DO
	IF IsNone(HasTagOption(_iEntity, 'Heating')) THEN
		CONTINUE;
	END_IF
	
	IF IsOk(GetReceiver(_iEntity, '*._onRequest', _iRec)) THEN
		IF IsErr(_ctx.priv.iRequestEvent.Pair(_iRec), nOut => _r) THEN
			DebugMsg(_iRec, strb.Append('Cannot pair _onRequest with this receiver! Error code: ').Append(TO_STRING(_r)).Read());
		END_IF
		
		RETURN;
	END_IF
END_WHILE

DebugMsg(THIS^, strb.Append('Cannot pair _requestEvent with a ').Append('_onRequest').Append('!').Read());
DebugMsg(_iEntity, strb.Append('_onRequest').Append(' not found!').Read());
END_METHOD

METHOD PROTECTED OnEntry
_ctx.io.bOpenValves := FALSE;

_ctx.priv.bActive := TRUE;
_ctx.priv.bReady := FALSE;

_ctx.hmi.sStatusText := 'Heating ON: Low Temperature...';
_ctx.hmi.nStatusColor := COL.BLACK.Raw;

_ctx.hmi.bHideReset := TRUE;

_ctx.priv.iRequestEvent.Emit(_ctx);
END_METHOD

METHOD PROTECTED OnExecute
IF _ctx.hmi.bDisable THEN
	_ctx.state.iMgr.Request(_ctx.state.iDisable);
ELSIF _rTemperature >= _hmi.rHighTemperature THEN
	_ctx.priv.bReady := TRUE;
END_IF
END_METHOD

END_FUNCTION_BLOCK

// ---- Room/State/DemandHeating/Room_State_DemandHeating.TcPOU
FUNCTION_BLOCK Room_State_DemandHeating EXTENDS _Room_State IMPLEMENTS I_Execute
VAR
	_exe				: Execute(THIS^);
	_hmi				: Room_State_DemandHeating_Hmi;
	_tonActive			: TON;
END_VAR

METHOD PROTECTED CanActivate : BOOL
CanActivate := _ctx.state.iMgr.Current = _ctx.state.iIdle;
END_METHOD

METHOD Execute
VAR_INPUT
	nPhase: INT;
END_VAR
VAR
	_iSelf		: I_State := THIS^;
	_strb		: Strb;
END_VAR
_strb.Set(_ctx.hmi.sData)
		.Append(' On: ').Append(strf.SimpleTime(_tonActive.ET, 'S', 'M'));

_ctx.hmi.sData := _strb.Read();

IF _ctx.state.iMgr.Current <> _ctx.state.iIdle THEN
	RETURN;
END_IF

IF _ctx.state.iMgr.Current = _iSelf THEN
	RETURN;
END_IF

IF _hmi.bDemandButton THEN
	_ctx.state.iMgr.Request(THIS^);
END_IF
END_METHOD

METHOD Init
VAR
	i			: Iter(1);
	_iEntity	: I_Entity;
	_iRec		: I_Receiver;
	_r			: Result;
	strb		: Strb;
END_VAR
WHILE IsOk(GetEntity(i.Next(), _iEntity)) DO
	IF IsNone(HasTagOption(_iEntity, 'Heating')) THEN
		CONTINUE;
	END_IF
	
	IF IsOk(GetReceiver(_iEntity, '*._onRequest', _iRec)) THEN
		IF IsErr(_ctx.priv.iRequestEvent.Pair(_iRec), nOut => _r) THEN
			DebugMsg(_iRec, strb.Append('Cannot pair _onRequest with this receiver! Error code: ').Append(TO_STRING(_r)).Read());
		END_IF
		
		RETURN;
	END_IF
END_WHILE

DebugMsg(THIS^, strb.Append('Cannot pair _requestEvent with a ').Append('_onRequest').Append('!').Read());
DebugMsg(_iEntity, strb.Append('_onRequest').Append(' not found!').Read());
END_METHOD

METHOD PROTECTED OnEntry
_ctx.io.bOpenValves := FALSE;

_ctx.priv.bActive := TRUE;
_ctx.priv.bReady := FALSE;

_ctx.hmi.sStatusText := 'Heating ON: Scheduled demand...';
_ctx.hmi.nStatusColor := COL.BLACK.Raw;

_ctx.hmi.bHideReset := TRUE;

_tonActive(IN := FALSE);

_ctx.priv.iRequestEvent.Emit(_ctx);
END_METHOD

METHOD PROTECTED OnExecute
_tonActive(IN := _ctx.io.bValvesOpen, PT := UDINT_TO_TIME(_hmi.nActivationTime * 1000));
IF _ctx.hmi.bDisable THEN
	_ctx.state.iMgr.Request(_ctx.state.iDisable);
ELSIF NOT _hmi.bDemandButton THEN
	_ctx.priv.bReady := TRUE;
ELSIF _tonActive.Q THEN
	_ctx.priv.bReady := TRUE;
	_hmi.bDemandButton := FALSE;
END_IF
END_METHOD

METHOD PROTECTED OnExit
VAR_INPUT
END_VAR
_hmi.bDemandButton := FALSE;
END_METHOD

END_FUNCTION_BLOCK

// ---- Room/Rooms/ReceptionRoom.TcPOU
FUNCTION_BLOCK ReceptionRoom EXTENDS BaseRoom
VAR_INPUT
	rTemperature	: LREAL := 20.0 + Math.Random();
END_VAR
VAR    
    // Entity
    _entityExtend	: EntityExtend(_entityStart);
	
    _lowTemperature	: Room_State_LowTemperature(_ctx, rTemperature);
	
    _entityEnd2		: EntityEnd;
END_VAR

METHOD Execute
VAR_INPUT
	nPhase: INT;
END_VAR
SUPER^.Execute(nPhase);

// Simulation
IF NOT sim.bTick THEN
	RETURN;
END_IF

IF bInletValve AND bOutletValve THEN
	rTemperature := rTemperature + sim.param.rRoomTemperatureRisePerHeater * Math.Random();
END_IF

rTemperature := rTemperature + sim.param.rRoomTemperaturePassiveDrop * Math.Random();

IF rTemperature < 0 THEN
	rTemperature := 0;
ELSIF rTemperature > 100 THEN
	rTemperature := 100;
END_IF
END_METHOD

END_FUNCTION_BLOCK

// ---- MAIN/SIM/Tick.TcPOU
FUNCTION Tick : BOOL
VAR_INPUT
	nTimeInMs	: ULINT;
	nTaskInMs	: ULINT := 20;
END_VAR

Tick := (GetSysTime() MOD (nTimeInMs * 10_000)) < (nTaskInMs * 10_000);

END_FUNCTION

// ---- GlobalTextList.TcGTLO
TEXTLIST GlobalTextList
  443 = '%.2f'
  858 = '%2.2f'
  701 = '%2.2f bar'
  165 = '%2.2f bar/tick'
  1000 = '%2.2f min'
  388 = '%2.2f s'
  181 = '%2.2f °C'
  899 = '%2.2f °C/tick'
  252 = '%i'
  752 = '%i min'
  296 = '%i s'
  862 = '%s'
  231 = 'Active'
  553 = 'Auto Sim'
  595 = 'Burner'
  999 = 'Burner Overload'
  870 = 'Click to change'
  18 = 'Demand'
  819 = 'Demand Activation Time'
  935 = 'Demand Active'
  969 = 'Drain Outlet Open'
  754 = 'Drain Outlet Valve Open'
  445 = 'Drain Speed: %.4f'
  336 = 'Enable Switch'
  958 = 'Enable Tank Switch'
  520 = 'EStop Button'
  707 = 'Feedback Ok'
  476 = 'Fill Speed: %.4f'
  923 = 'Filling Timeout:'
  698 = 'Filling Timeout: %s'
  393 = 'Heating'
  226 = 'Heating:'
  371 = 'High Level: %.2f'
  140 = 'High Level: %s'
  42 = 'High Temperature'
  254 = 'hmi.sMultiButtonText'
  89 = 'Level Sensor'
  616 = 'Low Level: %.2f'
  234 = 'Low Level: %s'
  738 = 'Low Temperature'
  762 = 'Max Pressure'
  409 = 'Max Pressure:'
  676 = 'Max Temp.'
  397 = 'Max Temp.:'
  731 = 'Mid Temp.'
  67 = 'Mid Temp.:'
  141 = 'Min Pressure'
  32 = 'Min Pressure:'
  630 = 'Min Temp.'
  441 = 'Min Temp.:'
  700 = 'NoWater'
  848 = 'OFF Delay'
  934 = 'ON delay'
  998 = 'Overload'
  728 = 'PASSIVE HEATING'
  116 = 'Press to Reset'
  342 = 'Pump'
  317 = 'Pump Overload'
  190 = 'Request Button'
  261 = 'Request Level: %.2f'
  452 = 'Request Level: %s'
  160 = 'Reset Output'
  106 = 'Room'
  64 = 'RoomTemperaturePassiveDrop'
  649 = 'RoomTemperatureRisePerHeater'
  111 = 'rRoomTemperaturePassiveDrop'
  468 = 'rRoomTemperatureRisePerHeater'
  142 = 'rSystemPressureFall'
  531 = 'rSystemPressureRise'
  247 = 'rSystemTemperatureDropPassive'
  485 = 'rSystemTemperatureDropPerHeater'
  498 = 'rSystemTemperatureFall'
  155 = 'rSystemTemperatureRise'
  173 = 'rSystemTemperatureRisePerBurner'
  305 = 'Run Output'
  300 = 'RunPump'
  489 = 'Safety'
  684 = 'Safety Ok'
  444 = 'Safety Run'
  517 = 'SafetyOk'
  629 = 'Simulation'
  411 = 'State:'
  587 = 'State: %s'
  664 = 'Status:'
  233 = 'Status: %s'
  471 = 'Sys. Pressure.'
  974 = 'Sys. Pressure.:'
  548 = 'Sys. Temp.'
  446 = 'Sys. Temp.:'
  338 = 'System Operational'
  534 = 'SystemPressureFall'
  450 = 'SystemPressureRise'
  420 = 'SystemTemperatureDropPassive'
  410 = 'SystemTemperatureDropPerHeater'
  648 = 'SystemTemperatureFall'
  264 = 'SystemTemperatureRise'
  918 = 'SystemTemperatureRisePerBurner'
  12 = 'Tank 0'
  237 = 'Tank 1'
  741 = 'Tank 2'
  288 = 'Tank 3'
  262 = 'Tick'
  743 = 'Timeout'
  737 = 'Timeout: %.2f'
  430 = 'Timeout: %s'
  596 = 'Toggle'
  315 = 'ToggleValveFault'
  379 = 'ToggleValveFault - Next valve action will fail'
  1064 = 'ToggleValveFault - Next valve actuation will fail'
  168 = 'TriggerValveFault'
END_TEXTLIST

// ---- MAIN/MAIN.TcVIS
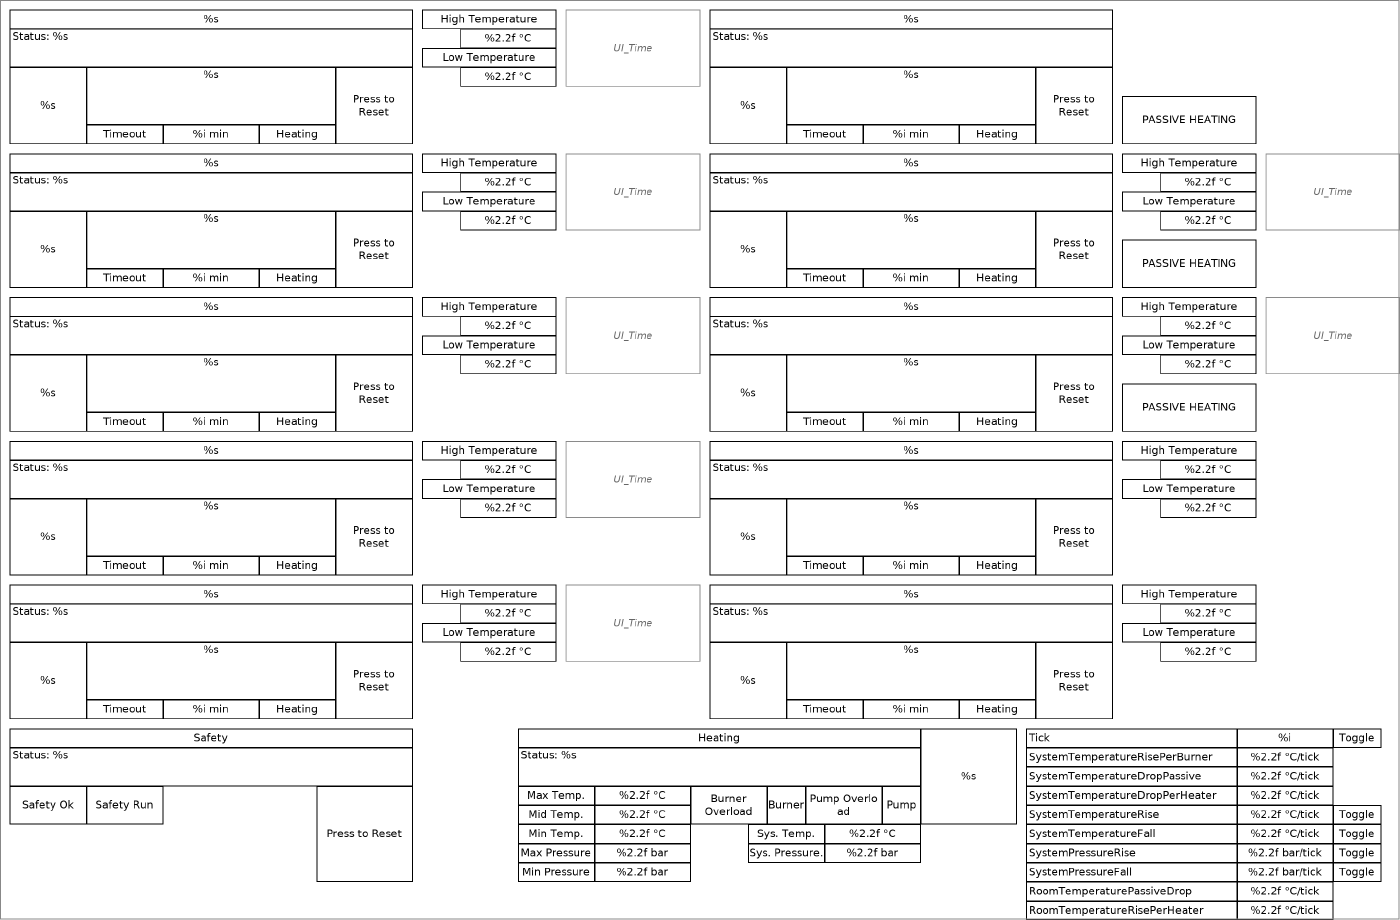
VISUALIZATION MAIN  // 1460x960
    Frame (10,760 520x100)
        shows UI_Safety(pou := MAIN.safety)
    Frame (540,760 520x160)
        shows UI_Heating(pou := MAIN.heating)
    Frame (10,10 420x140)
        shows UI_Room(ctx := MAIN.standardRoom[1]._ctx)
    Frame (10,160 420x140)
        shows UI_Room(ctx := MAIN.standardRoom[2]._ctx)
    Frame (10,310 420x140)
        shows UI_Room(ctx := MAIN.standardRoom[3]._ctx)
    Frame (10,460 420x140)
        shows UI_Room(ctx := MAIN.standardRoom[4]._ctx)
    Frame (10,610 420x140)
        shows UI_Room(ctx := MAIN.standardRoom[5]._ctx)
    Frame (440,10 140x80)
        shows UI_Temp(setting := MAIN.standardRoom[1]._settings.temp)
    Frame (440,160 140x80)
        shows UI_Temp(setting := MAIN.standardRoom[2]._settings.temp)
    Frame (440,310 140x80)
        shows UI_Temp(setting := MAIN.standardRoom[3]._settings.temp)
    Frame (440,460 140x80)
        shows UI_Temp(setting := MAIN.standardRoom[4]._settings.temp)
    Frame (440,610 140x80)
        shows UI_Temp(setting := MAIN.standardRoom[5]._settings.temp)
    Frame (740,10 420x140)
        shows UI_Room(ctx := MAIN.receptionRoom._ctx)
    Frame (740,160 420x140)
        shows UI_Room(ctx := MAIN.conferentionRoom01._ctx)
    Frame (740,310 420x140)
        shows UI_Room(ctx := MAIN.conferentionRoom02._ctx)
    Frame (740,460 420x140)
        shows UI_Room(ctx := MAIN.storeRoom01._ctx)
    Frame (740,610 420x140)
        shows UI_Room(ctx := MAIN.storeRoom02._ctx)
    Frame (1170,160 140x80)
        shows UI_Temp(setting := MAIN.conferentionRoom01._settings.temp)
    Frame (1170,310 140x80)
        shows UI_Temp(setting := MAIN.conferentionRoom02._settings.temp)
    Frame (1170,460 140x80)
        shows UI_Temp(setting := MAIN.storeRoom01._settings)
    Frame (1170,610 140x80)
        shows UI_Temp(setting := MAIN.storeRoom02._settings)
    Frame (1320,160 140x80)
        shows UI_Time(settings := MAIN.conferentionRoom01._settings.timee)
    Frame (590,10 140x80)
        shows UI_Time(settings := MAIN.standardRoom[1]._settings.timee)
    Frame (590,160 140x80)
        shows UI_Time(settings := MAIN.standardRoom[2]._settings.timee)
    Frame (590,310 140x80)
        shows UI_Time(settings := MAIN.standardRoom[3]._settings.timee)
    Frame (590,610 140x80)
        shows UI_Time(settings := MAIN.standardRoom[5]._settings.timee)
    Frame (590,460 140x80)
        shows UI_Time(settings := MAIN.standardRoom[4]._settings.timee)
    Frame (1320,310 140x80)
        shows UI_Time(settings := MAIN.conferentionRoom02._settings.timee)
    Rectangle (1170,400 140x50), "PASSIVE HEATING", colour toggle: MAIN.conferentionRoom02._settings.bEnablePassive
        toggle MAIN.conferentionRoom02._settings.bEnablePassive
    Rectangle (1170,250 140x50), "PASSIVE HEATING", colour toggle: MAIN.conferentionRoom01._settings.bEnablePassive
        toggle MAIN.conferentionRoom01._settings.bEnablePassive
    Rectangle (1170,100 140x50), "PASSIVE HEATING"
        toggle MAIN.receptionRoom._bEnablePassive
    Frame (1070,760 370x200)
        shows UI_Sim(param := SIM.param)
END_VISUALIZATION

// ---- _UI/UI_Heating.TcVIS
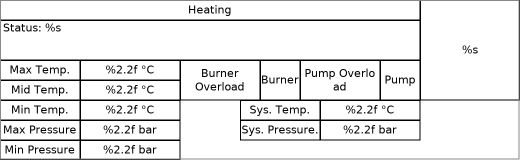
VISUALIZATION UI_Heating  // 520x160
VAR_IN_OUT
	pou			: Heating<CST.MAX_ROOM>;
END_VAR
VAR
END_VAR
    Rectangle (0,0 420x20), "Heating"
    Rectangle (0,20 420x40), "Status: %s", text variable: pou._ctx.hmi.sStatusText
        p55702900: pou._ctx.hmi.nStatusColor
    Rectangle (420,0 100x100), "%s", text variable: pou._ctx.hmi.sButtonText
        p55702900: pou._ctx.hmi.nButtonColor
        toggle pou._ctx.hmi.bButton
    Rectangle (0,60 80x20), "Max Temp."
    Rectangle (0,80 80x20), "Mid Temp."
    Rectangle (0,100 80x20), "Min Temp."
    Rectangle (80,60 100x20), "%2.2f °C", text variable: pou._ctx.hmi.rMaxTemperature
        OnMouseClick: write the text variable via Default
    Rectangle (80,80 100x20), "%2.2f °C", text variable: pou._ctx.hmi.rStdTemperature
        OnMouseClick: write the text variable via Default
    Rectangle (80,100 100x20), "%2.2f °C", text variable: pou._ctx.hmi.rMinTemperature
        OnMouseClick: write the text variable via Default
    Rectangle (0,140 80x20), "Min Pressure"
    Rectangle (0,120 80x20), "Max Pressure"
    Rectangle (80,120 100x20), "%2.2f bar", text variable: pou._ctx.hmi.rMaxPressure
        OnMouseClick: write the text variable via Default
    Rectangle (80,140 100x20), "%2.2f bar", text variable: pou._ctx.hmi.rMinPressure
        OnMouseClick: write the text variable via Default
    Rectangle (380,60 40x40), "Pump", colour toggle: pou.bPump
        toggle pou.bPump
    Rectangle (260,60 40x40), "Burner", colour toggle: pou.bBurner
        toggle pou.bBurner
    Rectangle (300,60 80x40), "Pump Overload", colour toggle: pou.bPumpOverload
        toggle pou.bPumpOverload
    Rectangle (180,60 80x40), "Burner Overload", colour toggle: pou.bBurnerOverload
        toggle pou.bBurnerOverload
    Rectangle (320,120 100x20), "%2.2f bar", text variable: pou.rBoilerPressure
    Rectangle (240,100 80x20), "Sys. Temp."
    Rectangle (240,120 80x20), "Sys. Pressure."
    Rectangle (320,100 100x20), "%2.2f °C", text variable: pou.rBoilerTemp
END_VISUALIZATION

// ---- _UI/UI_Safety.TcVIS
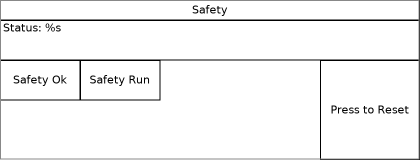
VISUALIZATION UI_Safety  // 420x160
VAR_IN_OUT
	pou			: Safety<CST.MAX_ESTOP>;
END_VAR
    Rectangle (0,0 420x20), "Safety"
    Rectangle (0,20 420x40), "Status: %s", text variable: pou._hmi.sStatusText
        p55702900: pou._hmi.nStatusColor
    Rectangle (320,60 100x100), "Press to Reset", invisible if: pou._hmi.bHideReset
        toggle pou._hmi.bReset
    Rectangle (0,60 80x40), "Safety Ok", colour toggle: pou.bSafetyOk
        toggle pou.bSafetyOk
    Rectangle (80,60 80x40), "Safety Run", colour toggle: pou.bSafetyRun
        toggle pou.bSafetyRun
END_VISUALIZATION

// ---- _UI/UI_Room.TcVIS
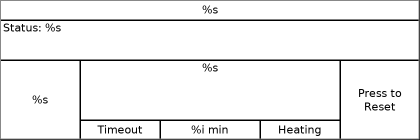
VISUALIZATION UI_Room  // 420x140
VAR_IN_OUT
	ctx			: Room_Ctx;
END_VAR
    Rectangle (0,0 420x20), "%s", text variable: CONCAT('Room ', UDINT_TO_STRING(ctx.hmi.nId))
    Rectangle (0,20 420x40), "Status: %s", text variable: ctx.hmi.sStatusText
        p55702900: ctx.hmi.nStatusColor
    Rectangle (0,60 80x80), "%s", text variable: ctx.hmi.sDisableText
        toggle ctx.hmi.bDisable
    Rectangle (340,60 80x80), "Press to Reset", invisible if: ctx.hmi.bHideReset
        toggle ctx.hmi.bReset
    Rectangle (80,60 260x60), "%s", text variable: ctx.hmi.sData
    Rectangle (160,120 100x20), "%i min", text variable: ctx.hmi.nTimeout
        OnMouseClick: write the text variable via Default
    Rectangle (80,120 80x20), "Timeout"
    Rectangle (260,120 80x20), "Heating", colour toggle: ctx.io.bValvesOpen
END_VISUALIZATION

// ---- _UI/UI_Sim.TcVIS
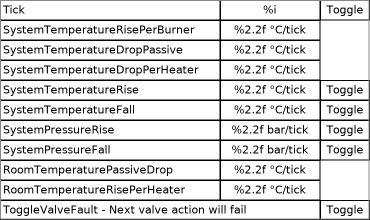
VISUALIZATION UI_Sim  // 370x220
VAR_IN_OUT
	param			: SimulationGlobalParameters;
END_VAR
    Rectangle (220,40 100x20), "%2.2f °C/tick", text variable: param.rSystemTemperatureDropPassive
        OnMouseClick: write the text variable via Default
    Rectangle (0,20 220x20), "SystemTemperatureRisePerBurner"
    Rectangle (220,20 100x20), "%2.2f °C/tick", text variable: param.rSystemTemperatureRisePerBurner
        OnMouseClick: write the text variable via Default
    Rectangle (0,40 220x20), "SystemTemperatureDropPassive"
    Rectangle (0,60 220x20), "SystemTemperatureDropPerHeater"
    Rectangle (0,80 220x20), "SystemTemperatureRise"
    Rectangle (0,100 220x20), "SystemTemperatureFall"
    Rectangle (0,120 220x20), "SystemPressureRise"
    Rectangle (0,140 220x20), "SystemPressureFall"
    Rectangle (0,160 220x20), "RoomTemperaturePassiveDrop"
    Rectangle (0,180 220x20), "RoomTemperatureRisePerHeater"
    Rectangle (220,80 100x20), "%2.2f °C/tick", text variable: param.rSystemTemperatureRise
        OnMouseClick: write the text variable via Default
    Rectangle (220,60 100x20), "%2.2f °C/tick", text variable: param.rSystemTemperatureDropPerHeater
        OnMouseClick: write the text variable via Default
    Rectangle (220,120 100x20), "%2.2f bar/tick", text variable: param.rSystemPressureRise
        OnMouseClick: write the text variable via Default
    Rectangle (220,100 100x20), "%2.2f °C/tick", text variable: param.rSystemTemperatureFall
        OnMouseClick: write the text variable via Default
    Rectangle (220,160 100x20), "%2.2f °C/tick", text variable: param.rRoomTemperaturePassiveDrop
        OnMouseClick: write the text variable via Default
    Rectangle (220,140 100x20), "%2.2f bar/tick", text variable: param.rSystemPressureFall
        OnMouseClick: write the text variable via Default
    Rectangle (220,180 100x20), "%2.2f °C/tick", text variable: param.rRoomTemperatureRisePerHeater
        OnMouseClick: write the text variable via Default
    Rectangle (0,0 220x20), "Tick"
    Rectangle (220,0 100x20), "%i", text variable: param.nTick
        OnMouseClick: write the text variable via Default
    Rectangle (320,80 50x20), "Toggle", colour toggle: param.bToggleSystemTemperatureRise
        toggle param.bToggleSystemTemperatureRise
    Rectangle (320,100 50x20), "Toggle", colour toggle: param.bToggleSystemTemperatureFall
        toggle param.bToggleSystemTemperatureFall
    Rectangle (320,120 50x20), "Toggle", colour toggle: param.bToggleSystemPressureRise
        toggle param.bToggleSystemPressureRise
    Rectangle (320,140 50x20), "Toggle", colour toggle: param.bToggleSystemPressureFall
        toggle param.bToggleSystemPressureFall
    Rectangle (320,0 50x20), "Toggle", colour toggle: param.bToggleSim
        toggle param.bToggleSim
    Rectangle (0,200 320x20), "ToggleValveFault - Next valve action will fail"
    Rectangle (320,200 50x20), "Toggle", colour toggle: param.bToggleValveFault
        toggle param.bToggleValveFault
END_VISUALIZATION

// ---- _UI/UI_Temp.TcVIS
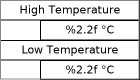
VISUALIZATION UI_Temp  // 140x80
VAR_IN_OUT
	setting		: Room_Settings_TemperatureSettings;
END_VAR
    Rectangle (0,40 140x20), "Low Temperature"
    Rectangle (40,60 100x20), "%2.2f °C", text variable: setting.rLow
        OnMouseClick: write the text variable via Default
    Rectangle (0,0 140x20), "High Temperature"
    Rectangle (40,20 100x20), "%2.2f °C", text variable: setting.rHigh
        OnMouseClick: write the text variable via Default
END_VISUALIZATION
